FUNCTION_BLOCK MachadoSFC (* Composite Function Block Type *)
  (* Standard: 61499-2 *)
  (* Version 0.2, 2003-12-05, JHC, Rockwell Automation, Renamed from NEWCOMPFB. *)
  (* Version 0.1, 2002-01-08, JHC, Rockwell Automation, Added DLY FB as example. *)
  (* Version 0.0, 2000-05-27, JHC, Rockwell Automation *)
  (* Compiler header: package fb.rt.pnp; *)
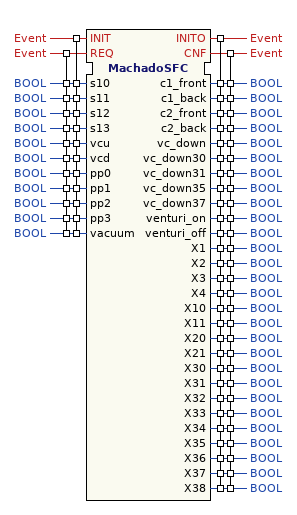
  EVENT_INPUT
    INIT WITH s10, s11, s13, s12, vcu, vcd, pp0, pp1, pp2, pp3, vacuum;
    REQ WITH s10, s11, s12, s13, vcu, vcd, pp0, pp1, pp2, pp3, vacuum; (* Normal Execution Request *)
  END_EVENT
  EVENT_OUTPUT
    INITO WITH c1_front, c1_back, c2_front, c2_back, vc_down, venturi_on, venturi_off, X1, X2, X3, X4, X10, X11, X20, X21, X30, X31, X32, X33, X34, X35, X36, X37, X38, vc_down30, vc_down31, vc_down35, vc_down37;
    CNF WITH c1_front, c1_back, c2_front, c2_back, vc_down, venturi_on, venturi_off, X1, X2, X3, X4, X10, X11, X20, X21, X30, X31, X32, X33, X34, X35, X36, X37, X38, vc_down30, vc_down31, vc_down35, vc_down37; (* Execution Confirmation *)
  END_EVENT
  VAR_INPUT
    s10 : BOOL; (* Input event qualifier *)
    s11 : BOOL;
    s12 : BOOL;
    s13 : BOOL;
    vcu : BOOL;
    vcd : BOOL;
    pp0 : BOOL;
    pp1 : BOOL;
    pp2 : BOOL;
    pp3 : BOOL;
    vacuum : BOOL;
  END_VAR
  VAR_OUTPUT
    c1_front : BOOL; (* Output event qualifier *)
    c1_back : BOOL;
    c2_front : BOOL;
    c2_back : BOOL;
    vc_down : BOOL;
    vc_down30 : BOOL;
    vc_down31 : BOOL;
    vc_down35 : BOOL;
    vc_down37 : BOOL;
    venturi_on : BOOL;
    venturi_off : BOOL;
    X1 : BOOL;
    X2 : BOOL;
    X3 : BOOL;
    X4 : BOOL;
    X10 : BOOL;
    X11 : BOOL;
    X20 : BOOL;
    X21 : BOOL;
    X30 : BOOL;
    X31 : BOOL;
    X32 : BOOL;
    X33 : BOOL;
    X34 : BOOL;
    X35 : BOOL;
    X36 : BOOL;
    X37 : BOOL;
    X38 : BOOL;
  END_VAR
  FBS
    SFC1 : SFC1;
    SFC2 : SFC2;
    SFC3 : SFC2;
    SFC4 : SFC4;
  END_FBS
  EVENT_CONNECTIONS
    INIT TO SFC1.INIT;
    REQ TO SFC1.REQ;
    SFC1.CNF TO SFC2.REQ;
    SFC3.CNF TO CNF;
    SFC2.CNF TO CNF;
    SFC1.INITO TO SFC2.INIT;
    SFC2.INITO TO SFC3.INIT;
    SFC3.INITO TO SFC4.INIT;
    SFC3.CNF TO SFC4.REQ;
    SFC2.CNF TO SFC4.REQ;
    SFC4.INITO TO INITO;
    SFC4.CNF TO CNF;
    SFC4.CNF TO SFC2.REQ;
    SFC4.CNF TO SFC1.REQ;
    REQ TO SFC4.REQ;
    REQ TO SFC3.REQ;
    SFC1.CNF TO SFC3.REQ;
    REQ TO SFC2.REQ;
  END_CONNECTIONS
  DATA_CONNECTIONS
    pp1 TO SFC1.pp1;
    pp2 TO SFC1.pp2;
    pp3 TO SFC1.pp3;
    s12 TO SFC3.s12;
    s13 TO SFC3.s3;
    SFC1.X2 TO SFC3.X12;
    SFC1.X3 TO SFC3.X3;
    SFC1.X1 TO SFC2.X12;
    s13 TO SFC2.s3;
    SFC1.X3 TO SFC2.X3;
    s10 TO SFC4.s0;
    s11 TO SFC4.s1;
    s12 TO SFC4.s2;
    s13 TO SFC4.s3;
    SFC1.X1 TO SFC4.X1;
    SFC1.X2 TO SFC4.X2;
    SFC1.X3 TO SFC4.X3;
    SFC2.CGO TO SFC4.X11;
    SFC3.CGO TO SFC4.X21;
    pp0 TO SFC4.pp0;
    vcu TO SFC4.vcu;
    vcd TO SFC4.vcd;
    vacuum TO SFC4.vacuum;
    SFC2.CGO TO c1_front;
    SFC3.CGO TO c2_front;
    SFC4.L1CGI TO c1_back;
    SFC4.L2CGI TO c2_back;
    SFC1.X1 TO X1;
    SFC1.X2 TO X2;
    SFC1.X3 TO X3;
    SFC4.X30 TO SFC3.X30;
    SFC4.X30 TO SFC2.X30;
    SFC4.vc_down30 TO vc_down30;
    SFC4.vc_down31 TO vc_down31;
    SFC4.vc_down35 TO vc_down35;
    SFC4.vc_down37 TO vc_down37;
    SFC4.venturi_on TO venturi_on;
    SFC4.venturi_off TO venturi_off;
    SFC4.X30 TO X30;
    SFC4.X31 TO X31;
    SFC4.X32 TO X32;
    SFC4.X33 TO X33;
    SFC4.X34 TO X34;
    SFC4.X35 TO X35;
    SFC4.X36 TO X36;
    SFC4.X37 TO X37;
    SFC4.X38 TO X38;
    SFC4.VCGD TO vc_down;
    SFC1.X4 TO X4;
    SFC2.X11 TO X11;
    SFC3.X10 TO X20;
    SFC3.X11 TO X21;
    SFC2.X10 TO X10;
    s11 TO SFC2.s12;
  END_CONNECTIONS
END_FUNCTION_BLOCK
